PROGRAM PRG_MachineLogger
VAR CONSTANT
	sMACHINE_LOGGER_NAME		: STRING := 'PMS';
	sMACHINE_LOGGER_DIRECTORY	: STRING := '\Hard Disk\';
	sMACHINE_LOGGER_FILE_NAME	: STRING := 'Machine_Logger_';
END_VAR
VAR
	bFirstCycle : BOOL	:= TRUE; (* Auxilary bit for initial setup assignaments *)
	bTestWrite : BOOL;
	bActivated : BOOL; 
END_VAR

IF bFirstCycle THEN
	bFirstCycle := FALSE;
	fbMachineLogger.MR_FirstCycle(	sName 			:= sMACHINE_LOGGER_NAME,
									sFileDir		:= sMACHINE_LOGGER_DIRECTORY,
									sFileName 		:= sMACHINE_LOGGER_FILE_NAME,
									sAmsNetId 		:= '',
									bAddTimeStamp	:= TRUE,
									bAddHeader		:= TRUE);

	

END_IF

IF NOT fbMachineLogger.Active THEN
	fbMachineLogger.MR_Init();
END_IF
(* Cyclic run *)
fbMachineLogger();
IF bTestWrite THEN
	bTestWrite := 0;
	fbMachineLogger.MR_AddLogs( sLogMessage := 'this is test add log');
END_IF

END_PROGRAM

(* stored: Version 1.1.0.1, ProductVersion 3.1.4024.12
   POU PRG_MachineLogger: Id {2f1915c6-1e69-4780-a036-9c83e91b8a81}, SpecialFunc None *)
